(* CoDeSys 2.3.9.62 project: Cap11_13.pro *)
(* Libraries: Standard.lib 2.6.14 10:37:46, IecSfc.lib 2.6.14 10:37:46 *)

(* Global variable list: Global_Variables *)
VAR_GLOBAL

	(* Entradas *)
       M: BOOL;
 	P: BOOL;
	Rear: BOOL;
	L1: BOOL;
	L2: BOOL;
	FC: BOOL;

	(* Salidas*)
	 S1:BOOL;
       S2:BOOL;
       S3:BOOL;
END_VAR

(* POU PLC_PRG, CFC *)
PROGRAM PLC_PRG
VAR
END_VAR
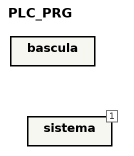
_CFC_ (* Continuous Function Chart, elements in execution order *)
#0 bascula()
#1 sistema()
_END_CFC_
(* the same logic as Structured Text *)
bascula();
sistema();
END_PROGRAM

(* POU bascula, SFC *)
PROGRAM bascula
VAR

END_VAR
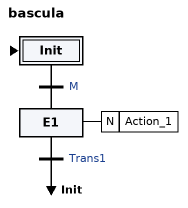
INITIAL_STEP Init:
END_STEP
TRANSITION FROM Init TO E1 := M;
END_TRANSITION
STEP E1:
	Action_1(N);
END_STEP
TRANSITION FROM E1 TO Init := Trans1;
END_TRANSITION
END_PROGRAM

(* POU sistema, ST *)
PROGRAM sistema
VAR
  peso:REAL;
  piston:REAL;
END_VAR
IF S1=TRUE AND S2=TRUE THEN
   peso:=peso+0.1;
ELSE
  IF S2=TRUE THEN
    peso:=peso+0.02;
  END_IF
END_IF

IF peso>5.9 AND peso<6.2 THEN
  L1:=TRUE;
ELSE
  L1:=FALSE;
END_IF

IF peso>9.9 THEN
  L2:=TRUE;
ELSE
  L2:=FALSE;
END_IF



IF S3=TRUE THEN
  piston:=piston+0.5;
END_IF

IF piston=10 THEN
   FC:=TRUE;
   peso:=0;
   piston:=0;
ELSE
   FC:=FALSE;
END_IF
END_PROGRAM

(* Visualisation Bascula
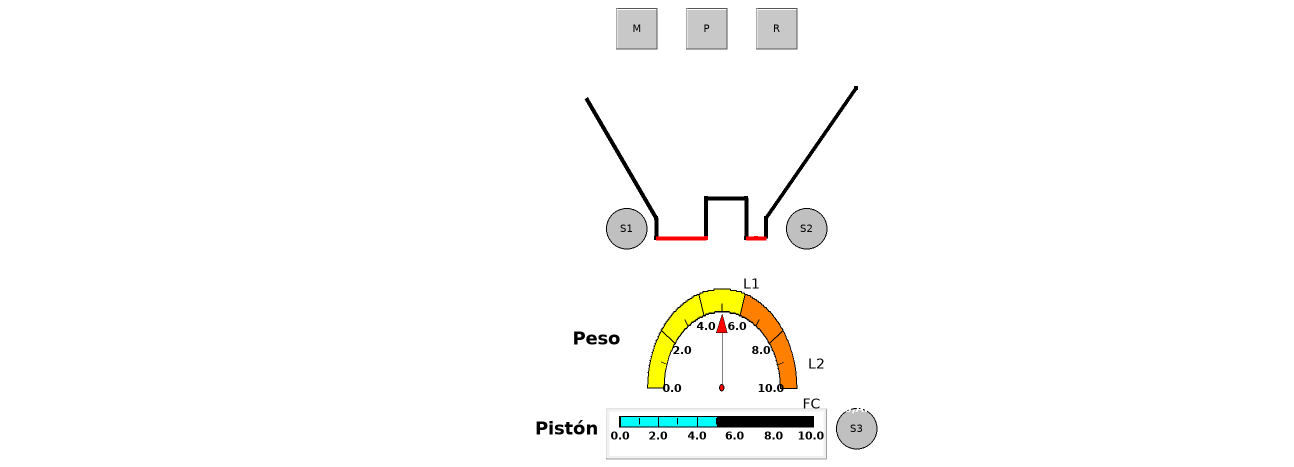
button at (100,50)-(141,91): text "M"; taps M
button at (170,50)-(211,91): text "P"; taps P
button at (240,50)-(281,91): text "R"; taps Rear
ellipse at (90,250)-(131,291): text "S1"; alarm colour if S1
ellipse at (270,250)-(311,291): text "S2"; alarm colour if S2
ellipse at (320,450)-(361,491): text "S3"; alarm colour if S3
polyline at (140,280)-(190,280): invisible if S1
polyline at (230,280)-(250,280): invisible if S2
group at (130,330)-(281,441)
  rectangle at (0,0)-(1,1): text "{ExtendedElement},Visu\ElementDLL.ete,0,@Zeigerinstrument,151,180,0,0,255,0,0,0,sistema.peso,,%.1f,1,1,1,1,2,0,10,0,0,0,0,0,0,0,-13,16,700,Arial,1,2,0,6,255,255,0,6,10,255,128,0,0,255,255,255,,0,0,0,0,"
  rectangle at (15,68)-(37,84): text "0.0"
  rectangle at (25,39)-(47,55): text "2.0"
  rectangle at (49,21)-(71,37): text "4.0"
  rectangle at (80,21)-(102,37): text "6.0"
  rectangle at (104,39)-(126,55): text "8.0"
  rectangle at (110,68)-(139,84): text "10.0"
  polygon at (70,20)-(81,76): angle ((sistema.peso * 1.0)-5) * 18
group at (90,450)-(311,501)
  rectangle at (0,0)-(1,1): text "{ExtendedElement},Visu\ElementDLL.ete,1,@Bargraph,221,51,1,0,0,sistema.piston,,%.1f,1,2,0,10,0,0,0,0,0,0,0,-13,16,700,Arial,0,255,255,255,0,0,0,0,1,1,0,0,0,,0,0,0,"
  rectangle at (14,9)-(111,18): alarm colour if (sistema.piston) < 0; right ((sistema.piston * 1.0) - 5)  * 19.2
  rectangle at (2,20)-(26,47): text "0.0"
  rectangle at (40,20)-(64,47): text "2.0"
  rectangle at (79,20)-(103,47): text "4.0"
  rectangle at (117,20)-(141,47): text "6.0"
  rectangle at (156,20)-(180,47): text "8.0"
  rectangle at (189,20)-(222,47): text "10.0"
rectangle at (40,350)-(121,411): text "Peso"
rectangle at (220,310)-(251,341): text "L1"; alarm colour if L1
rectangle at (290,390)-(311,421): text "L2"; alarm colour if L2
rectangle at (10,440)-(91,501): text "Pistón"
rectangle at (280,430)-(311,461): text "FC"; alarm colour if FC
39 more shapes without text or variables
*)
